FUNCTION_BLOCK Outfeed EXTENDS FB_PackML_BaseModule
VAR
	CurrentCustomMode : E_PMLCustomMode;
END_VAR

METHOD CyclicLogic
IF NOT _InitComplete THEN
	_InitComplete := Initialize();
	RETURN;
END_IF

CurrentCustomMode := _CurrentMode;

//
SUPER^.CyclicLogic();
END_METHOD

END_FUNCTION_BLOCK

(* stored: Version 1.1.0.1
   POU Outfeed: Id {281e2777-2c03-497a-82e3-651ecf3118b5}, SpecialFunc None
   Method CyclicLogic: Id {8aa2815e-daa4-4613-ada7-de5e6513f6c5} *)
